// TIA Portal V17 export
// export: Created 2025-03-05T07:59:28.3245828Z, ExportSetting WithDefaults, DisplayName Totally Integrated Automation Portal, DisplayVersion V17 Update 8, DisplayName TIA Portal Openness, DisplayVersion V17 Update 8, DisplayName TIA Portal Version Control Interface, DisplayVersion V17, DisplayName SINAMICS Startdrive Advanced, DisplayVersion V17 SP2, DisplayName SINAMICS Startdrive G110M, G120, G120C, G120D, G120P, G115D, DisplayVersion V17 SP2, DisplayName SINAMICS Startdrive G130, G150, S120, S150, SINAMICS MV, S210, DisplayVersion V17 SP2, DisplayName STEP 7 Professional, DisplayVersion V17 Update 8, DisplayName SINUMERIK ONE STEP 7 Toolbox, DisplayVersion V17 Update 12, DisplayName SINUMERIK 840D sl STEP 7 Toolbox, DisplayVersion V17 Update 12, DisplayName STEP 7 Safety, DisplayVersion V17 Update 6, DisplayName WinCC Advanced, DisplayVersion V17 Update 8
DATA_BLOCK "DB8000_PART_STATUS"   // DB8000
{ S7_Optimized_Access := 'FALSE'; DB_Accessible_From_OPC_UA := 'FALSE' }
AUTHOR : ETXETAR
VERSION : 1.0
// stored: AutoNumber false, DBAccessibleFromOPCUA false, DBAccessibleFromWebserver true, IsOnlyStoredInLoadMemory false, IsWriteProtectedInAS false
   VAR RETAIN
      HMI : Struct
         ONE_PART_LOADED_FOR_MACH : Bool;   // ONE PART LOADED FOR MACH
         UNIT_01_PART_PRESENT : Bool;   // HMI UNIT 01 PART PRESENT BUTTON
         UNIT_01_REMOVE_PART : Bool;   // HMI UNIT 01 REMOVE PART BUTTON
         UNIT_01_GOOD_PART : Bool;   // HMI UNIT 01 GOOD PART NOT MACHINED BUTTON
         UNIT_01_REJECT_PART : Bool;   // HMI UNIT 01 NOT OK PART BUTTON
         UNIT_01_MASTER_PART : Bool;   // HMI UNIT 01 SET MASTER PART
         UNIT_02_PART_PRESENT : Bool;   // HMI UNIT 02 PART PRESENT BUTTON
         UNIT_02_REMOVE_PART : Bool;   // HMI UNIT 02 REMOVE PART BUTTON
         UNIT_02_GOOD_PART : Bool;   // HMI UNIT 02 GOOD PART NOT MACHINED BUTTON
         UNIT_02_REJECT_PART : Bool;   // HMI UNIT 02 NOT OK PART BUTTON
         UNIT_02_MASTER_PART : Bool;   // HMI UNIT 02 SET MASTER PART
         UNIT_03_PART_PRESENT : Bool;   // HMI UNIT 03 PART PRESENT BUTTON
         UNIT_03_REMOVE_PART : Bool;   // HMI UNIT 03 REMOVE PART BUTTON
         UNIT_03_GOOD_PART : Bool;   // HMI UNIT 03 GOOD PART NOT MACHINED BUTTON
         UNIT_03_REJECT_PART : Bool;   // HMI UNIT 03 NOT OK PART BUTTON
         UNIT_03_MASTER_PART : Bool;   // HMI UNIT 03 SET MASTER PART
         PART_STATUS_FIXTURES_LIST : Int := 1;   // HMI PART STATUS FIXTURES LIST
         PART_STATUS_PART_TYPE_LIST : Int := 1;   // HMI PART STATUS PART TYPE LIST
         PART_STATUS_PART_STATUS_LIST : Int := 1;   // HMI PART STATUS PROCESS PART STATUS LIST
         PART_NUMBER_LIST : Int;   // PART TYPE LIST AUX
      END_STRUCT;
      UNIT_01 : Struct
         FIXTURE_1 : Struct
            PART_A { S7_SetPoint := 'True'} : "PART_STATUS_CLADDING";
         END_STRUCT;
         FIXTURE_2 : Struct
            PART_A { S7_SetPoint := 'True'} : "PART_STATUS_CLADDING";
         END_STRUCT;
         FIXTURE_3 : Struct
            PART_A { S7_SetPoint := 'True'} : "PART_STATUS_CLADDING";
         END_STRUCT;
         FIXTURE_4 : Struct
            PART_A { S7_SetPoint := 'True'} : "PART_STATUS_CLADDING";
         END_STRUCT;
         STATION_1 : Struct
            PART_A { S7_SetPoint := 'True'} : "PART_STATUS_CLADDING";
         END_STRUCT;
         STATION_2 : Struct
            PART_A { S7_SetPoint := 'True'} : "PART_STATUS_CLADDING";
         END_STRUCT;
         STATION_3 : Struct
            PART_A { S7_SetPoint := 'True'} : "PART_STATUS_CLADDING";
         END_STRUCT;
         STATION_4 : Struct
            PART_A { S7_SetPoint := 'True'} : "PART_STATUS_CLADDING";
         END_STRUCT;
      END_STRUCT;
      UNIT_02 : Struct
         FIXTURE_1 : Struct
            PART_A { S7_SetPoint := 'True'} : "PART_STATUS_CLADDING";
         END_STRUCT;
         FIXTURE_2 : Struct
            PART_A { S7_SetPoint := 'True'} : "PART_STATUS_CLADDING";
         END_STRUCT;
         FIXTURE_3 : Struct
            PART_A { S7_SetPoint := 'True'} : "PART_STATUS_CLADDING";
         END_STRUCT;
         FIXTURE_4 : Struct
            PART_A { S7_SetPoint := 'True'} : "PART_STATUS_CLADDING";
         END_STRUCT;
         STATION_1 : Struct
            PART_A { S7_SetPoint := 'True'} : "PART_STATUS_CLADDING";
         END_STRUCT;
         STATION_2 : Struct
            PART_A { S7_SetPoint := 'True'} : "PART_STATUS_CLADDING";
         END_STRUCT;
         STATION_3 : Struct
            PART_A { S7_SetPoint := 'True'} : "PART_STATUS_CLADDING";
         END_STRUCT;
         STATION_4 : Struct
            PART_A { S7_SetPoint := 'True'} : "PART_STATUS_CLADDING";
         END_STRUCT;
      END_STRUCT;
      UNIT_03 : Struct
         FIXTURE_1 : Struct
            PART_A { S7_SetPoint := 'True'} : "PART_STATUS_CLADDING";
         END_STRUCT;
      END_STRUCT;
      PULSE_1 : Bool;   // PULSE 1
      PULSE_2 : Bool;   // PULSE 2
      PULSE_3 : Bool;   // PULSE 3
      PULSE_4 : Bool;   // PULSE 4
      PULSE_5 : Bool;   // PULSE 5
      PULSE_6 : Bool;   // PULSE 6
      PULSE_7 : Bool;   // PULSE 7
      PULSE_8 : Bool;   // PULSE 8
      PULSE_9 : Bool;   // PULSE 9
      PULSE_10 : Bool;   // PULSE 10
      PULSE_11 : Bool;   // PULSE 11
      PULSE_12 : Bool;   // PULSE 12
      PULSE_13 : Bool;   // PULSE 13
      PULSE_14 : Bool;   // PULSE 14
      PULSE_15 : Bool;   // PULSE 15
      PULSE_16 : Bool;   // PULSE 16
      PULSE_17 : Bool;   // PULSE 17
      PULSE_18 : Bool;   // PULSE 18
      PULSE_19 : Bool;   // PULSE 19
      PULSE_20 : Bool;   // PULSE 20
      PULSE_21 : Bool;   // PULSE 21
      PULSE_22 : Bool;   // PULSE 22
      PULSE_23 : Bool;   // PULSE 23
      PULSE_24 : Bool;   // PULSE 24
   END_VAR
BEGIN
END_DATA_BLOCK
